{attribute 'GeneratedUsingTerminal: EL9930-0000-0017'}
{attribute addProperty BoxType "EL9930-0000-0017"}
{attribute addProperty Id "A_0004_EL9930_0001_0017EL9930_2CDB4CAF4"}
{attribute addProperty CRC "1648505753"}
{attribute addProperty Size "4"}
TYPE A_0003_EL9930_0000_0017_62423399 EXTENDS EL9930_2C0891BD :
STRUCT
	{attribute addProperty Name "A_0004_EL9930_0001_0017"}
	{attribute addProperty PreviousPort "A_0003(EL9930-0000-0017) : B"}
	A_0004_EL9930_0001_0017 : EL9930_2CDB4CAF;
END_STRUCT
END_TYPE

(* stored: Version 1.2.0.0, ProductVersion 3.1.4024.9
   DUT A_0003_EL9930_0000_0017_62423399: Id {1d902255-8bdb-4388-8486-a0714c33d7ab} *)
